DATA_BLOCK "bioPID.DB"
{ S7_Optimized_Access := 'TRUE' }
VERSION : 1.0
// Batch I/O PID Data Block:
// by Woermann Automation
NON_RETAIN
   VAR RETAIN
      pid : Array[0..15] of "bioPID.DT";
   END_VAR

BEGIN

END_DATA_BLOCK

